PROGRAM P_CraneControl
VAR
 	fbStatus 					: FB_Status;
	fbRunningClock 				: FB_Clock;
	fbManualControl 			: FB_ManualControl; 
	bEnableManualControl 		: BOOL;
	fbAutomaticControl 			: FB_AutomaticControl;
	bEnableAutomaticControl 	: BOOL; 
	fbActiveDamping 			: FB_ActiveDamping;
	fControlOutputNormalized 	: LREAL; 
	
	ADtest0 : LREAL;
	ADtest1 : LREAL;
	ADtest2 : LREAL;
	ADtest : BOOL;
END_VAR

fbStatus(
bFault := G_Work.bFault,
eMode := G_Work.eMode,
fTime := fbRunningClock.fTime,
eStatus => G_Work.eStatus
);

fbRunningClock(
	bStart := (fbStatus.eStatus = E_Status.Starting) OR (fbStatus.eStatus = E_Status.Running),
	bStop := (fbStatus.eStatus = E_Status.Stopping),
	fCycleTime := G_Parameters.stParam.fCyclicTime
);

fbManualControl(
	eMode := G_Work.eMode,
	eStatus := G_Work.eStatus,
	stParam := G_Parameters.stParam, 
);

fbAutomaticControl(
	eMode := G_Work.eMode,
	eStatus := G_Work.eStatus,
	stAutomaticControlSettings := G_Commissioning.stAutomaticControlSettings,
	stMotionReferenceGeneratorSettings := G_Commissioning.stMotionReferenceGeneratorSettings,
	stParam := G_Parameters.stParam,
	fPositionFeedback := G_Sensors.fPistonPosition
);

fbActiveDamping(
	ssMethodType := BOOL_TO_SINT(G_Commissioning.stAutomaticControlSettings.bEnableActiveDamping),
	bEnable := (fbStatus.eStatus = E_Status.Running),
	stParam := G_Parameters.stParam,
	fPressurePistonSide_Pa := F_BarToEng(G_Sensors.fPressurePistonSide),
	fPressureRodSide_Pa := F_BarToEng(G_Sensors.fPressureRodSide)
);

IF (G_Work.eMode = E_Mode.Manual AND G_Work.eStatus = E_Status.Running) THEN
	fControlOutputNormalized := LIMIT(-1.0, (fbManualControl.fControlOutputNormalized - fbActiveDamping.fPressureFeedbackNormalized), 1.0);
ELSIF (G_Work.eMode = E_Mode.Auto AND G_Work.eStatus = E_Status.Running) THEN
	fControlOutputNormalized := LIMIT(-1.0, (-fbAutomaticControl.fControlOutputNormalized - fbActiveDamping.fPressureFeedbackNormalized), 1.0);
ELSE
	fControlOutputNormalized := 0.0;
END_IF

//G_Work.fControlOutputNormalized := fControlOutputNormalized;

END_PROGRAM

(* stored: Version 1.1.0.1, ProductVersion 3.1.4024.13
   POU P_CraneControl: Id {c8d14843-0c4e-4243-a583-0726f2828bd5}, SpecialFunc None *)
